// TwinCAT 3 PLC project PLC
// ProgramVersion: 3.1.4024.0
// libraries:
//   Tc2_MC2, * (Beckhoff Automation GmbH)
//   Tc2_Standard, * (Beckhoff Automation GmbH)
//   Tc2_System, * (Beckhoff Automation GmbH)
//   Tc3_Module, * (Beckhoff Automation GmbH)
//   Triamec EtherCAT Lib, * (Triamec Motion AG)
// project tree:
//   GVLs/ Triamec_GVL.TcGVL
//   / PlcTask.TcTTO
//   POUs/ DriveControlledHoming.TcPOU, MAIN.TcPOU, NC_Axis.TcPOU
// real-time tasks:
//   TASK PlcTask: cycle T#10ms, priority 20, ADS port 350
// motion (NC):
//   TASK NC-Task 1 SAF: cycle T#2ms, priority 4, ADS port 501
//   TASK NC-Task 1 SVB: cycle T#10ms, priority 8, ADS port 511
//   AXIS Axis 1 (id 1)
//     OtherSettings: AllowMotionCmdToSlave=true
//     encoder EncType=19
//       EncPara: ScaleFactorNumerator=1e-06, MaxCount=#xffffffff
//     drive DrvType=16
//       DrvPara: MaxCount=#xffffffff, DriveControlDWord=#x00020100
//         Analog: TorqueSetpointScale=10, ScaleFactorActTorque=0.1
//         TimeComp: TaskDelayCycles=1
//     controller CtrType=9
//       CtrPara: PriorControlFactor=1
//         Observer: BandWidth=20
//   AXIS Axis 2 (id 2)
//     OtherSettings: AllowMotionCmdToSlave=true
//     encoder EncType=19
//       EncPara: ScaleFactorNumerator=1e-06, MaxCount=#xffffffff
//     drive DrvType=16
//       DrvPara: MaxCount=#xffffffff, DriveControlDWord=#x00020100
//         Analog: TorqueSetpointScale=10, ScaleFactorActTorque=0.1
//         TimeComp: TaskDelayCycles=1
//     controller CtrType=9
//       CtrPara: PriorControlFactor=1
//         Observer: BandWidth=20
// I/O:
//   DEVICE Device 1 (EtherCAT), AmsNetId 10.20.34.98.2.1
//     Drive 1 (TSD) [TSD_minFW4.22]
//       modules: Axis 0, Axis 0, Axis 0, Axis 0, Axis 0, Axis 1, Axis 1, Axis 1, Axis 1, Axis 1
// variable links:
//   NC-Task 1 SAF/Axes/Axis 1 <-> Device 1 (EtherCAT)/Drive 1 (TSD)
//     Drive/Inputs/In/nDataIn1 <-> Axis 0/PositionInputs/PositionError
//     Drive/Inputs/In/nDataIn3[0] <-> Axis 0/TorqueInputs/TorqueActual
//     Drive/Inputs/In/nDcOutputTime <-> InfoData/DcOutputShift
//     Drive/Inputs/In/nState1 <-> Axis 0/MainInputs/Status Word
//     Drive/Inputs/In/nState2 <-> Axis 0/MainInputs/Status Word @bit 8
//     Drive/Inputs/In/nState4 @bit 1 <-> WcState/InputToggle
//     Drive/Inputs/In/nState4 <-> WcState/WcState
//     Drive/Inputs/In/nState5 <-> Axis 0/MainInputs/Mode of Operation Display
//     Drive/Outputs/Out/nCtrl1 <-> Axis 0/MainOutputs/Control Word
//     Drive/Outputs/Out/nCtrl2 <-> Axis 0/MainOutputs/Control Word @bit 8
//     Drive/Outputs/Out/nCtrl5 <-> Axis 0/MainOutputs/Mode of Operation
//     Drive/Outputs/Out/nDataOut1 <-> Axis 0/PositionOutputs/TargetPosition
//     Drive/Outputs/Out/nDataOut2 <-> Axis 0/VelocityOutputs/TargetVelocity
//     Drive/Outputs/Out/nDataOut4[0] <-> Axis 0/TorqueOutputs/TargetTorque
//     Enc/Inputs/In/nDataIn1 <-> Axis 0/MainInputs/ActualPosition
//     Enc/Inputs/In/nDataIn7 <-> Axis 0/VelocityInputs/ActualVelocity
//     Enc/Inputs/In/nDcInputTime <-> InfoData/DcInputShift
//     Enc/Inputs/In/nState4 @bit 1 <-> WcState/InputToggle
//     Enc/Inputs/In/nState4 <-> WcState/WcState
//   NC-Task 1 SAF/Axes/Axis 2 <-> Device 1 (EtherCAT)/Drive 1 (TSD)
//     Drive/Inputs/In/nDataIn1 <-> Axis 1/PositionInputs/PositionError
//     Drive/Inputs/In/nDataIn3[0] <-> Axis 1/TorqueInputs/TorqueActual
//     Drive/Inputs/In/nDcOutputTime <-> InfoData/DcOutputShift
//     Drive/Inputs/In/nState1 <-> Axis 1/MainInputs/Status Word
//     Drive/Inputs/In/nState2 <-> Axis 1/MainInputs/Status Word @bit 8
//     Drive/Inputs/In/nState4 @bit 1 <-> WcState/InputToggle
//     Drive/Inputs/In/nState4 <-> WcState/WcState
//     Drive/Inputs/In/nState5 <-> Axis 1/MainInputs/Mode of Operation Display
//     Drive/Outputs/Out/nCtrl1 <-> Axis 1/MainOutputs/Control Word
//     Drive/Outputs/Out/nCtrl2 <-> Axis 1/MainOutputs/Control Word @bit 8
//     Drive/Outputs/Out/nCtrl5 <-> Axis 1/MainOutputs/Mode of Operation
//     Drive/Outputs/Out/nDataOut1 <-> Axis 1/PositionOutputs/TargetPosition
//     Drive/Outputs/Out/nDataOut2 <-> Axis 1/VelocityOutputs/TargetVelocity
//     Drive/Outputs/Out/nDataOut4[0] <-> Axis 1/TorqueOutputs/TargetTorque
//     Enc/Inputs/In/nDataIn1 <-> Axis 1/MainInputs/ActualPosition
//     Enc/Inputs/In/nDataIn7 <-> Axis 1/VelocityInputs/ActualVelocity
//     Enc/Inputs/In/nDcInputTime <-> InfoData/DcInputShift
//     Enc/Inputs/In/nState4 @bit 1 <-> WcState/InputToggle
//     Enc/Inputs/In/nState4 <-> WcState/WcState
//   PLC/PLC Instance <-> NC-Task 1 SAF/Axes/Axis 1
//     PlcTask Inputs/MAIN.Axis[0].ncRef.NcToPlc <-> Outputs/ToPlc
//     PlcTask Outputs/MAIN.Axis[0].ncRef.PlcToNc <-> Inputs/FromPlc
//   PLC/PLC Instance <-> NC-Task 1 SAF/Axes/Axis 2
//     PlcTask Inputs/MAIN.Axis[1].ncRef.NcToPlc <-> Outputs/ToPlc
//     PlcTask Outputs/MAIN.Axis[1].ncRef.PlcToNc <-> Inputs/FromPlc

CONFIGURATION PLC
    RESOURCE PLC ON TwinCAT3
        TASK PlcTask(INTERVAL := T#10ms, PRIORITY := 20);
        PROGRAM MAIN WITH PlcTask : MAIN;
    END_RESOURCE
END_CONFIGURATION

// ---- GVLs/Triamec_GVL.TcGVL

VAR_GLOBAL
	gEnableAxes			: BOOL;	(* variable to enable all axes *)
	gStatusAxesEnabled 	: BOOL;	(* variable indicates that all axes enabled *)
	gHoming				: BOOL; (* variable to execute drive controlled homing *)	
END_VAR

// ---- POUs/MAIN.TcPOU
PROGRAM MAIN
VAR
	Axis	: ARRAY [0..1] OF NC_Axis;
	axisIdx	: UINT;
END_VAR

(* configuration *)
Axis[0].config.driveId		:= 1001;				// Drive 1 (TSD)/EtherCAT/EtherCAT-Addr.
Axis[0].config.netId		:= '192.168.10.99.2.1';	// Drive 1 (TSD)^InfoData^AdsAddr^netId
Axis[0].config.axisNumber	:= 0;					// first (0) or second (1) axis of a dual axis drive
Axis[0].config.axisId		:= 0;					// cnc-axis-id used in events
Axis[0].refPos 				:= 0.14;				// reference position for drive controlled homing
Axis[1].config.driveId		:= 1001;				// Drive 1 (TSD)/EtherCAT/EtherCAT-Addr.
Axis[1].config.netId		:= '192.168.10.99.2.1';	// Drive 1 (TSD)^InfoData^AdsAddr^netId
Axis[1].config.axisNumber	:= 1;					// first (0) or second (1) axis of a dual axis drive
Axis[1].config.axisId		:= 1;					// cnc-axis-id used in events
Axis[1].refPos 				:= 0.09;				// reference position for drive controlled homing

(* Axis handler *)
FOR axisIdx := 0 TO SIZEOF(Axis)/SIZEOF(Axis[0])-1 DO
	Axis[axisIdx].enable := gEnableAxes;
	Axis[axisIdx].home := gHoming;
	Axis[axisIdx]();
	IF NOT Axis[axisIdx].enabled THEN
		gStatusAxesEnabled := FALSE;
	END_IF
END_FOR

END_PROGRAM

// ---- POUs/NC_Axis.TcPOU
FUNCTION_BLOCK NC_Axis EXTENDS TE_AxisBase0
VAR_INPUT
	enable		: BOOL;
	reset		: BOOL;
	home		: BOOL;
	refPos		: LREAL;
END_VAR
VAR_OUTPUT
	ready		: BOOL;
	enabled		: BOOL;
	referenced	: BOOL;
	error		: BOOL;
END_VAR
VAR
	ncRef		: AXIS_REF;
	ncPower		: MC_Power;
	ncReset		: MC_Reset;
	drvHoming	: DriveControlledHoming;
END_VAR


ncPower.Enable			:= enable;
ncPower.Enable_Negative	:= TRUE;
ncPower.Enable_Positive	:= TRUE;
ncPower(Axis:= ncRef);

ncReset.Execute := reset;
ncReset(Axis := ncRef);

ncRef.ReadStatus();

enabled := ncRef.Status.ControlLoopClosed AND ncRef.Status.Operational;
referenced := ncRef.Status.Homed;
error := ncRef.Status.Error;

(* drive controlled homing *)
drvHoming.execute := home;
drvHoming.refPos := refPos;
drvHoming(axis := THIS^, axisRef := ncRef);

(* This handles errors (error=TRUE) and warnings (error=FALSE) as TwinCat message *)
CallSlow();

END_FUNCTION_BLOCK

// ---- POUs/DriveControlledHoming.TcPOU
FUNCTION_BLOCK DriveControlledHoming
VAR_IN_OUT
	axis 		: TE_AxisBase0;
	axisRef 	: AXIS_REF;
END_VAR
VAR_INPUT
	execute 	: BOOL;
	refPos		: LREAL;
END_VAR
VAR_OUTPUT
	error 		: BOOL;
	done		: BOOL;
END_VAR
VAR
	writeReg	: TE_RegisterWriteInt32;
	ncOpMode	: MC_WriteDriveOperationMode;
	ncHome		: MC_Home;
	ncReset		: MC_Reset;
	writeRef	: TE_RegisterWriteFloat64;
	driveStatus : NCTOPLC_AXIS_REF_STATE2;
	timeout     : INT := 0;
	state		: INT := 0;
END_VAR

// Sample code for drive controlled homing of an axis
// configure homing in the TAM System Explorer using registers Axes[].Parameters.Homing
// Refer to application note AN141 Homing Procedures and Setup
// Use the standard mode of operation HM=6 of the EtherCAT CoE standard
// or the following sample code, which overcomes NC position reset after homing

driveStatus := axisRef.NcToPlc.StateDWord2;

CASE state OF
	0:  // Idle
		done	:= FALSE;
		error	:= FALSE;
		IF execute THEN
			writeRef(axis:=axis, execute := FALSE);
			timeout := 0;
			state := state + 10;
		END_IF
		
	10:  // write reference position
		// The user might want to avoid writing the position here, if he wants to use the value set in the startup menu
		IF axis.config.axisNumber = 0 THEN
			writeRef.address	:= 16#23EE00;
		ELSE
			writeRef.address	:= 16#2BEE00; // offset 0x800 for second axis
		END_IF
		writeRef(axis:=axis, execute:=TRUE, value:=refPos);
		IF NOT execute THEN
			state	:= 999;
		ELSIF writeRef.done THEN
			writeRef(axis:=axis, execute:=FALSE);
			ncHome(Axis:=axisRef, Execute := FALSE);
			timeout := 0;
			state	:= state + 10;
		ELSIF writeRef.error THEN
			error := TRUE;
		END_IF
	
	20:	// enter homing mode of operation  
		// NC_Home does not seem to support drive controlled homing
		// To start drive controlled homing, we change to modeOfOperation 6 and
		// then we use the fact, that the ControlWord flag 0x10 is already set.
		// This starts homing in the drive which causes the homing done flag 15 turned off
		timeout := timeout + 1;
		ncOpMode.Execute := TRUE;
		ncOpMode.DriveOperationMode := E_DriveOperationMode.DriveOperationMode_DriveBasedHoming;
		IF NOT execute THEN
			state := 999;
		ELSIF axis.messageId <> 0 THEN
			error		:= TRUE;
		ELSIF ncOpMode.Done AND (driveStatus.Value AND 16#8000) = 0 THEN
			writeReg(axis:=axis, execute := FALSE);
			state := state + 10;
		ELSIF timeout>10 THEN 
			// The modeOfOperation should change within 0.1ms and the homing flag should disappear within another 0.1 ms
			// Possible causes for this error are: The controlWord 0x10 flag is not set because the NC shows an error
			error := TRUE;
		END_IF

	30:	// wait for homing finished
		IF NOT execute THEN
			// user commanded an abort
			// since the axis might be moving, we have to stop homing first
			writeReg.value		:= 2; // stop homing enum RCTeHoC_Stop
			IF axis.config.axisNumber = 0 THEN
				writeReg.address	:= 16#23EC00;
			ELSE
				writeReg.address	:= 16#2BEC00; // offset 0x800 for second axis
			END_IF
			writeReg(axis:=axis, execute := TRUE);
			state		:= state + 10;
		ELSIF axis.messageId <> 0 THEN
			error		:= TRUE;
		ELSIF (driveStatus.Value AND 16#8000) = 16#8000 THEN
			ncReset(Axis:=axisRef, Execute := FALSE);
			state		:= state + 20;
		END_IF

	40:	// wait for stop command finished (not the stopping itself)
		writeReg(axis:=axis, execute := TRUE);
		IF NOT execute THEN
			state	:= 999;
		ELSIF writeReg.done THEN
			IF writeReg.error THEN
				error	:= TRUE;
			ELSE
				writeReg(axis:=axis, execute := FALSE);
				state	:= 999;
			END_IF
		END_IF
		
	50:	// reset the NC to force Setpoint=Actual
		ncReset(Axis:=axisRef, Execute := TRUE);
		IF NOT execute THEN
			state	:= 999;
		ELSIF ncReset.Error OR axis.messageId<>0 THEN
			error	:= TRUE;
		ELSIF ncReset.Done THEN
			// wait some time for position settle before mode change to CSP (8)
			ncReset(Axis:=axisRef, Execute := FALSE);
			ncHome(Axis:=axisRef, Execute := FALSE);
			state	:= state + 10;
		END_IF
		
	60:	// write homing done to NC. This just sets the homing done bit in the NC
		ncHome.HomingMode := MC_HomingMode.MC_ForceCalibration;
		ncHome(Axis:=axisRef, Execute := TRUE);
		IF NOT execute THEN
			ncHome(Axis:=axisRef, Execute := FALSE);
			state	:= 999;
		ELSIF NOT ncHome.Busy THEN
			IF ncHome.Error THEN
				state := 999;
				error	:= TRUE;
			ELSE
				ncHome(Axis:=axisRef, Execute := FALSE);
				done	:= TRUE;
				state	:= 999; // homing finished
			END_IF
		END_IF
		
	999: // homing finished or error handling
		ncOpMode.Execute := TRUE;
		ncOpMode.DriveOperationMode := E_DriveOperationMode.DriveOperationMode_Pos1;
		IF ncOpMode.Error OR ncOpMode.Done AND NOT execute THEN
			ncOpMode.Execute := FALSE;
			done := FALSE;
			state := 0;	
		END_IF

ELSE
	state := 0;
END_CASE
ncOpMode(axis := axisRef);

END_FUNCTION_BLOCK
